// TIA Portal V16 export
// export: Created 2025-08-01T13:38:02.7356342Z, ExportSetting WithDefaults, DisplayName Totally Integrated Automation Portal, DisplayVersion V16, DisplayName TIA Portal Version Control Interface, DisplayVersion V16, DisplayName TIA Portal Openness, DisplayVersion V16, DisplayName STEP 7 Professional, DisplayVersion V16, DisplayName STEP 7 Safety, DisplayVersion V16, DisplayName WinCC Advanced, DisplayVersion V16
DATA_BLOCK "MC_Jog_OB1"   // DB56
VERSION : 0.1
// stored: AutoNumber true, InstanceOfName MC_Jog, InstanceOfType FB
"MC_Jog"
   // VAR_INPUT
   //    "Jog Forward" : Bool;
   //    "Jog Backward" : Bool;
   //    Speed : Int;
   //    Brake : Bool;
   // END_VAR
   // VAR_OUTPUT
   //    "Drive Fwd Output" : Bool;
   //    "Drive Rev Output" : Bool;
   //    "Drive Speed Output" : Int;
   //    "Drive Brake Output" : Bool;
   // END_VAR
BEGIN
END_DATA_BLOCK
